// TIA Portal V17 export
// export: Created 2025-03-07T09:17:03.08606Z, ExportSetting WithDefaults, DisplayName Totally Integrated Automation Portal, DisplayVersion V17 Update 8, DisplayName TIA Portal Openness, DisplayVersion V17 Update 8, DisplayName TIA Portal Version Control Interface, DisplayVersion V17, DisplayName SINAMICS Startdrive Advanced, DisplayVersion V17 SP2, DisplayName SINAMICS Startdrive G110M, G120, G120C, G120D, G120P, G115D, DisplayVersion V17 SP2, DisplayName SINAMICS Startdrive G130, G150, S120, S150, SINAMICS MV, S210, DisplayVersion V17 SP2, DisplayName STEP 7 Professional, DisplayVersion V17 Update 8, DisplayName SINUMERIK ONE STEP 7 Toolbox, DisplayVersion V17 Update 12, DisplayName SINUMERIK 840D sl STEP 7 Toolbox, DisplayVersion V17 Update 12, DisplayName STEP 7 Safety, DisplayVersion V17 Update 6, DisplayName WinCC Advanced, DisplayVersion V17 Update 8
FUNCTION "FC7451_QUALITY_ON_DEMAND_CLADDING" : Void   // FC7451, LAD
{ S7_Optimized_Access := 'FALSE' }
AUTHOR : ETXETAR
NAME : GM-QC
VERSION : 1.0
// stored: AutoNumber false, IsIECCheckEnabled false, SetENOAutomatically false, UDAEnableTagReadback false
   VAR CONSTANT
      FC_NUMBER : DInt := 7451;
   END_VAR
   VAR_TEMP   // added for the SCL form of the ladder/FBD networks
      _w1 : Bool;
      _w2 : Bool;
   END_VAR
BEGIN

REGION Network 1: //////////_UNIT_01_//////////
END_REGION

REGION Network 2: FIXTURE 1 PART A DEMAND SET
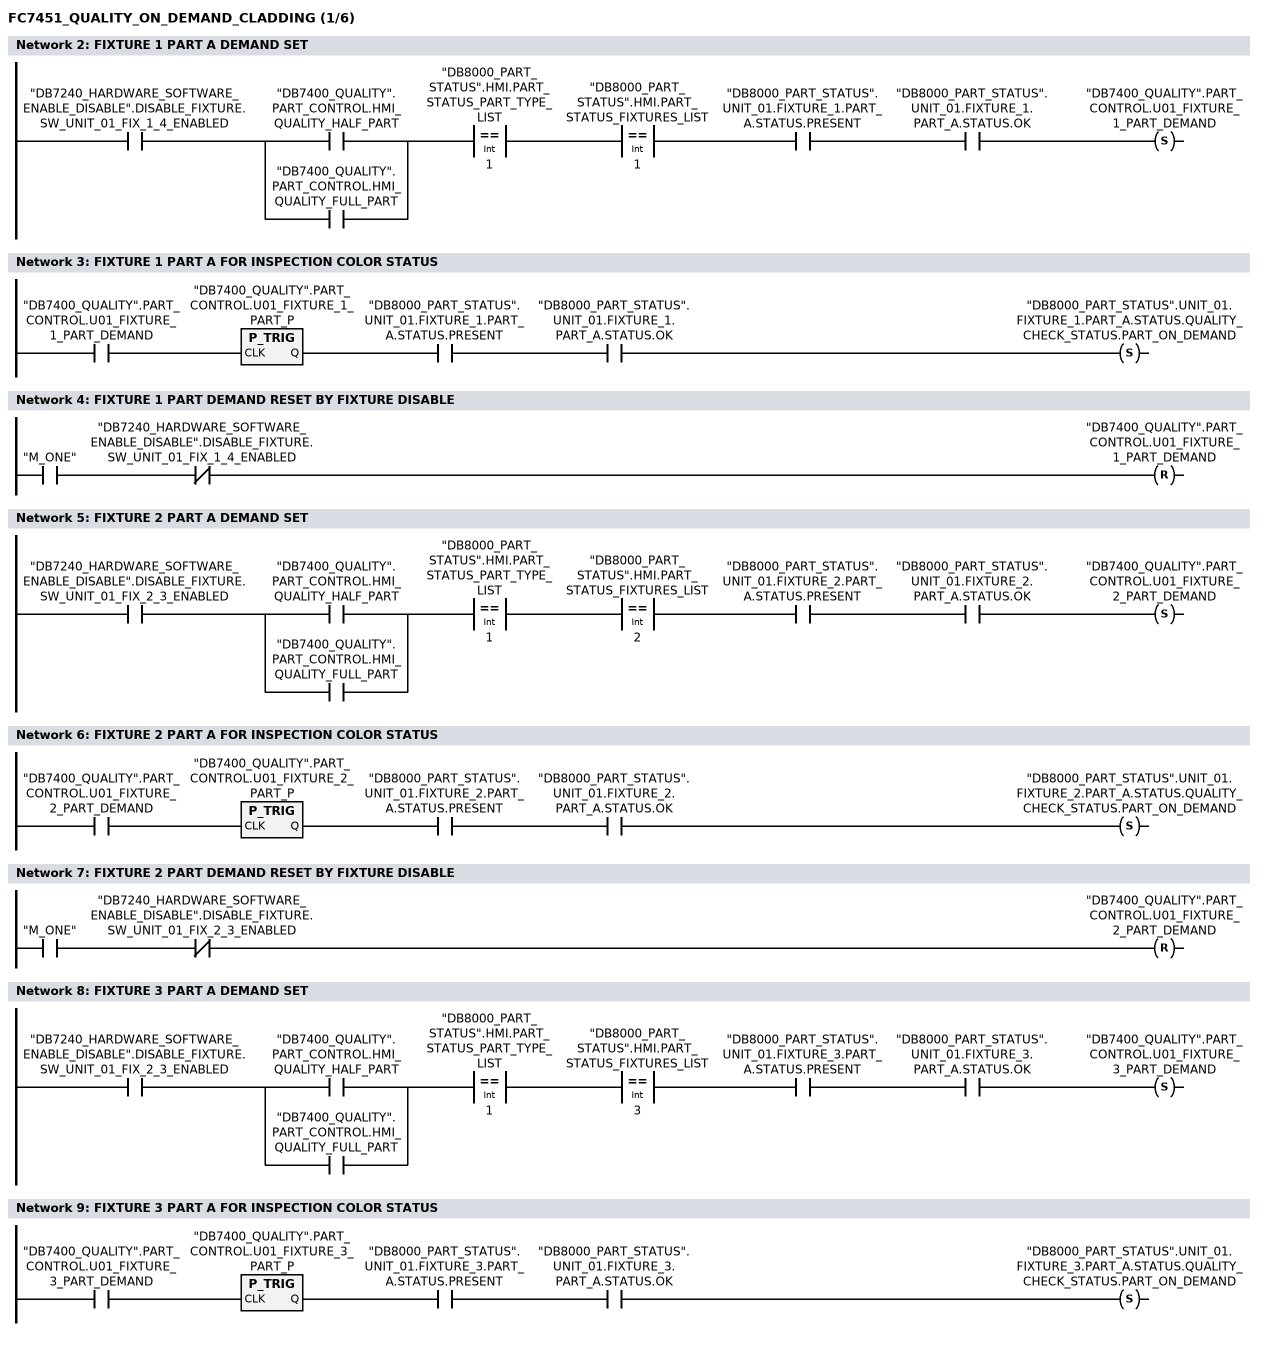
   RUNG wire#powerrail
      Contact( "DB7240_HARDWARE_SOFTWARE_ENABLE_DISABLE".DISABLE_FIXTURE.SW_UNIT_01_FIX_1_4_ENABLED )
      wire#w1
      Contact( "DB7400_QUALITY".PART_CONTROL.HMI_QUALITY_HALF_PART )
      wire#w2
      { S7_Templates := "SrcType := Int" } EQ_Contact(in1 := "DB8000_PART_STATUS".HMI.PART_STATUS_PART_TYPE_LIST, in2 := 1)
      { S7_Templates := "SrcType := Int" } EQ_Contact(in1 := "DB8000_PART_STATUS".HMI.PART_STATUS_FIXTURES_LIST, in2 := 1)
      Contact( "DB8000_PART_STATUS".UNIT_01.FIXTURE_1.PART_A.STATUS.PRESENT )
      Contact( "DB8000_PART_STATUS".UNIT_01.FIXTURE_1.PART_A.STATUS.OK )
      S_Coil( "DB7400_QUALITY".PART_CONTROL.U01_FIXTURE_1_PART_DEMAND )
   END_RUNG
   RUNG wire#w1
      Contact( "DB7400_QUALITY".PART_CONTROL.HMI_QUALITY_FULL_PART )
   END_RUNG wire#w2
   // the same network as SCL:
   IF "DB7240_HARDWARE_SOFTWARE_ENABLE_DISABLE".DISABLE_FIXTURE.SW_UNIT_01_FIX_1_4_ENABLED AND ("DB7400_QUALITY".PART_CONTROL.HMI_QUALITY_HALF_PART OR "DB7400_QUALITY".PART_CONTROL.HMI_QUALITY_FULL_PART) AND ("DB8000_PART_STATUS".HMI.PART_STATUS_PART_TYPE_LIST = 1) AND ("DB8000_PART_STATUS".HMI.PART_STATUS_FIXTURES_LIST = 1) AND "DB8000_PART_STATUS".UNIT_01.FIXTURE_1.PART_A.STATUS.PRESENT AND "DB8000_PART_STATUS".UNIT_01.FIXTURE_1.PART_A.STATUS.OK THEN
       "DB7400_QUALITY".PART_CONTROL.U01_FIXTURE_1_PART_DEMAND := TRUE;
   END_IF;
END_REGION

REGION Network 3: FIXTURE 1 PART A FOR INSPECTION COLOR STATUS
   RUNG wire#powerrail
      Contact( "DB7400_QUALITY".PART_CONTROL.U01_FIXTURE_1_PART_DEMAND )
      P_Trig( "DB7400_QUALITY".PART_CONTROL.U01_FIXTURE_1_PART_P )
      Contact( "DB8000_PART_STATUS".UNIT_01.FIXTURE_1.PART_A.STATUS.PRESENT )
      Contact( "DB8000_PART_STATUS".UNIT_01.FIXTURE_1.PART_A.STATUS.OK )
      S_Coil( "DB8000_PART_STATUS".UNIT_01.FIXTURE_1.PART_A.STATUS.QUALITY_CHECK_STATUS.PART_ON_DEMAND )
   END_RUNG
   // the same network as SCL:
   #_w1 := "DB7400_QUALITY".PART_CONTROL.U01_FIXTURE_1_PART_DEMAND AND NOT "DB7400_QUALITY".PART_CONTROL.U01_FIXTURE_1_PART_P;   // rising edge
   "DB7400_QUALITY".PART_CONTROL.U01_FIXTURE_1_PART_P := "DB7400_QUALITY".PART_CONTROL.U01_FIXTURE_1_PART_DEMAND;
   IF #_w1 AND "DB8000_PART_STATUS".UNIT_01.FIXTURE_1.PART_A.STATUS.PRESENT AND "DB8000_PART_STATUS".UNIT_01.FIXTURE_1.PART_A.STATUS.OK THEN
       "DB8000_PART_STATUS".UNIT_01.FIXTURE_1.PART_A.STATUS.QUALITY_CHECK_STATUS.PART_ON_DEMAND := TRUE;
   END_IF;
END_REGION

REGION Network 4: FIXTURE 1 PART DEMAND RESET BY FIXTURE DISABLE
   RUNG wire#powerrail
      Contact( "M_ONE" )
      I_Contact( "DB7240_HARDWARE_SOFTWARE_ENABLE_DISABLE".DISABLE_FIXTURE.SW_UNIT_01_FIX_1_4_ENABLED )
      R_Coil( "DB7400_QUALITY".PART_CONTROL.U01_FIXTURE_1_PART_DEMAND )
   END_RUNG
   // the same network as SCL:
   IF "M_ONE" AND NOT "DB7240_HARDWARE_SOFTWARE_ENABLE_DISABLE".DISABLE_FIXTURE.SW_UNIT_01_FIX_1_4_ENABLED THEN
       "DB7400_QUALITY".PART_CONTROL.U01_FIXTURE_1_PART_DEMAND := FALSE;
   END_IF;
END_REGION

REGION Network 5: FIXTURE 2 PART A DEMAND SET
   RUNG wire#powerrail
      Contact( "DB7240_HARDWARE_SOFTWARE_ENABLE_DISABLE".DISABLE_FIXTURE.SW_UNIT_01_FIX_2_3_ENABLED )
      wire#w1
      Contact( "DB7400_QUALITY".PART_CONTROL.HMI_QUALITY_HALF_PART )
      wire#w2
      { S7_Templates := "SrcType := Int" } EQ_Contact(in1 := "DB8000_PART_STATUS".HMI.PART_STATUS_PART_TYPE_LIST, in2 := 1)
      { S7_Templates := "SrcType := Int" } EQ_Contact(in1 := "DB8000_PART_STATUS".HMI.PART_STATUS_FIXTURES_LIST, in2 := 2)
      Contact( "DB8000_PART_STATUS".UNIT_01.FIXTURE_2.PART_A.STATUS.PRESENT )
      Contact( "DB8000_PART_STATUS".UNIT_01.FIXTURE_2.PART_A.STATUS.OK )
      S_Coil( "DB7400_QUALITY".PART_CONTROL.U01_FIXTURE_2_PART_DEMAND )
   END_RUNG
   RUNG wire#w1
      Contact( "DB7400_QUALITY".PART_CONTROL.HMI_QUALITY_FULL_PART )
   END_RUNG wire#w2
   // the same network as SCL:
   IF "DB7240_HARDWARE_SOFTWARE_ENABLE_DISABLE".DISABLE_FIXTURE.SW_UNIT_01_FIX_2_3_ENABLED AND ("DB7400_QUALITY".PART_CONTROL.HMI_QUALITY_HALF_PART OR "DB7400_QUALITY".PART_CONTROL.HMI_QUALITY_FULL_PART) AND ("DB8000_PART_STATUS".HMI.PART_STATUS_PART_TYPE_LIST = 1) AND ("DB8000_PART_STATUS".HMI.PART_STATUS_FIXTURES_LIST = 2) AND "DB8000_PART_STATUS".UNIT_01.FIXTURE_2.PART_A.STATUS.PRESENT AND "DB8000_PART_STATUS".UNIT_01.FIXTURE_2.PART_A.STATUS.OK THEN
       "DB7400_QUALITY".PART_CONTROL.U01_FIXTURE_2_PART_DEMAND := TRUE;
   END_IF;
END_REGION

REGION Network 6: FIXTURE 2 PART A FOR INSPECTION COLOR STATUS
   RUNG wire#powerrail
      Contact( "DB7400_QUALITY".PART_CONTROL.U01_FIXTURE_2_PART_DEMAND )
      P_Trig( "DB7400_QUALITY".PART_CONTROL.U01_FIXTURE_2_PART_P )
      Contact( "DB8000_PART_STATUS".UNIT_01.FIXTURE_2.PART_A.STATUS.PRESENT )
      Contact( "DB8000_PART_STATUS".UNIT_01.FIXTURE_2.PART_A.STATUS.OK )
      S_Coil( "DB8000_PART_STATUS".UNIT_01.FIXTURE_2.PART_A.STATUS.QUALITY_CHECK_STATUS.PART_ON_DEMAND )
   END_RUNG
   // the same network as SCL:
   #_w1 := "DB7400_QUALITY".PART_CONTROL.U01_FIXTURE_2_PART_DEMAND AND NOT "DB7400_QUALITY".PART_CONTROL.U01_FIXTURE_2_PART_P;   // rising edge
   "DB7400_QUALITY".PART_CONTROL.U01_FIXTURE_2_PART_P := "DB7400_QUALITY".PART_CONTROL.U01_FIXTURE_2_PART_DEMAND;
   IF #_w1 AND "DB8000_PART_STATUS".UNIT_01.FIXTURE_2.PART_A.STATUS.PRESENT AND "DB8000_PART_STATUS".UNIT_01.FIXTURE_2.PART_A.STATUS.OK THEN
       "DB8000_PART_STATUS".UNIT_01.FIXTURE_2.PART_A.STATUS.QUALITY_CHECK_STATUS.PART_ON_DEMAND := TRUE;
   END_IF;
END_REGION

REGION Network 7: FIXTURE 2 PART DEMAND RESET BY FIXTURE DISABLE
   RUNG wire#powerrail
      Contact( "M_ONE" )
      I_Contact( "DB7240_HARDWARE_SOFTWARE_ENABLE_DISABLE".DISABLE_FIXTURE.SW_UNIT_01_FIX_2_3_ENABLED )
      R_Coil( "DB7400_QUALITY".PART_CONTROL.U01_FIXTURE_2_PART_DEMAND )
   END_RUNG
   // the same network as SCL:
   IF "M_ONE" AND NOT "DB7240_HARDWARE_SOFTWARE_ENABLE_DISABLE".DISABLE_FIXTURE.SW_UNIT_01_FIX_2_3_ENABLED THEN
       "DB7400_QUALITY".PART_CONTROL.U01_FIXTURE_2_PART_DEMAND := FALSE;
   END_IF;
END_REGION

REGION Network 8: FIXTURE 3 PART A DEMAND SET
   RUNG wire#powerrail
      Contact( "DB7240_HARDWARE_SOFTWARE_ENABLE_DISABLE".DISABLE_FIXTURE.SW_UNIT_01_FIX_2_3_ENABLED )
      wire#w1
      Contact( "DB7400_QUALITY".PART_CONTROL.HMI_QUALITY_HALF_PART )
      wire#w2
      { S7_Templates := "SrcType := Int" } EQ_Contact(in1 := "DB8000_PART_STATUS".HMI.PART_STATUS_PART_TYPE_LIST, in2 := 1)
      { S7_Templates := "SrcType := Int" } EQ_Contact(in1 := "DB8000_PART_STATUS".HMI.PART_STATUS_FIXTURES_LIST, in2 := 3)
      Contact( "DB8000_PART_STATUS".UNIT_01.FIXTURE_3.PART_A.STATUS.PRESENT )
      Contact( "DB8000_PART_STATUS".UNIT_01.FIXTURE_3.PART_A.STATUS.OK )
      S_Coil( "DB7400_QUALITY".PART_CONTROL.U01_FIXTURE_3_PART_DEMAND )
   END_RUNG
   RUNG wire#w1
      Contact( "DB7400_QUALITY".PART_CONTROL.HMI_QUALITY_FULL_PART )
   END_RUNG wire#w2
   // the same network as SCL:
   IF "DB7240_HARDWARE_SOFTWARE_ENABLE_DISABLE".DISABLE_FIXTURE.SW_UNIT_01_FIX_2_3_ENABLED AND ("DB7400_QUALITY".PART_CONTROL.HMI_QUALITY_HALF_PART OR "DB7400_QUALITY".PART_CONTROL.HMI_QUALITY_FULL_PART) AND ("DB8000_PART_STATUS".HMI.PART_STATUS_PART_TYPE_LIST = 1) AND ("DB8000_PART_STATUS".HMI.PART_STATUS_FIXTURES_LIST = 3) AND "DB8000_PART_STATUS".UNIT_01.FIXTURE_3.PART_A.STATUS.PRESENT AND "DB8000_PART_STATUS".UNIT_01.FIXTURE_3.PART_A.STATUS.OK THEN
       "DB7400_QUALITY".PART_CONTROL.U01_FIXTURE_3_PART_DEMAND := TRUE;
   END_IF;
END_REGION

REGION Network 9: FIXTURE 3 PART A FOR INSPECTION COLOR STATUS
   RUNG wire#powerrail
      Contact( "DB7400_QUALITY".PART_CONTROL.U01_FIXTURE_3_PART_DEMAND )
      P_Trig( "DB7400_QUALITY".PART_CONTROL.U01_FIXTURE_3_PART_P )
      Contact( "DB8000_PART_STATUS".UNIT_01.FIXTURE_3.PART_A.STATUS.PRESENT )
      Contact( "DB8000_PART_STATUS".UNIT_01.FIXTURE_3.PART_A.STATUS.OK )
      S_Coil( "DB8000_PART_STATUS".UNIT_01.FIXTURE_3.PART_A.STATUS.QUALITY_CHECK_STATUS.PART_ON_DEMAND )
   END_RUNG
   // the same network as SCL:
   #_w1 := "DB7400_QUALITY".PART_CONTROL.U01_FIXTURE_3_PART_DEMAND AND NOT "DB7400_QUALITY".PART_CONTROL.U01_FIXTURE_3_PART_P;   // rising edge
   "DB7400_QUALITY".PART_CONTROL.U01_FIXTURE_3_PART_P := "DB7400_QUALITY".PART_CONTROL.U01_FIXTURE_3_PART_DEMAND;
   IF #_w1 AND "DB8000_PART_STATUS".UNIT_01.FIXTURE_3.PART_A.STATUS.PRESENT AND "DB8000_PART_STATUS".UNIT_01.FIXTURE_3.PART_A.STATUS.OK THEN
       "DB8000_PART_STATUS".UNIT_01.FIXTURE_3.PART_A.STATUS.QUALITY_CHECK_STATUS.PART_ON_DEMAND := TRUE;
   END_IF;
END_REGION

REGION Network 10: FIXTURE 3 PART DEMAND RESET BY FIXTURE DISABLE
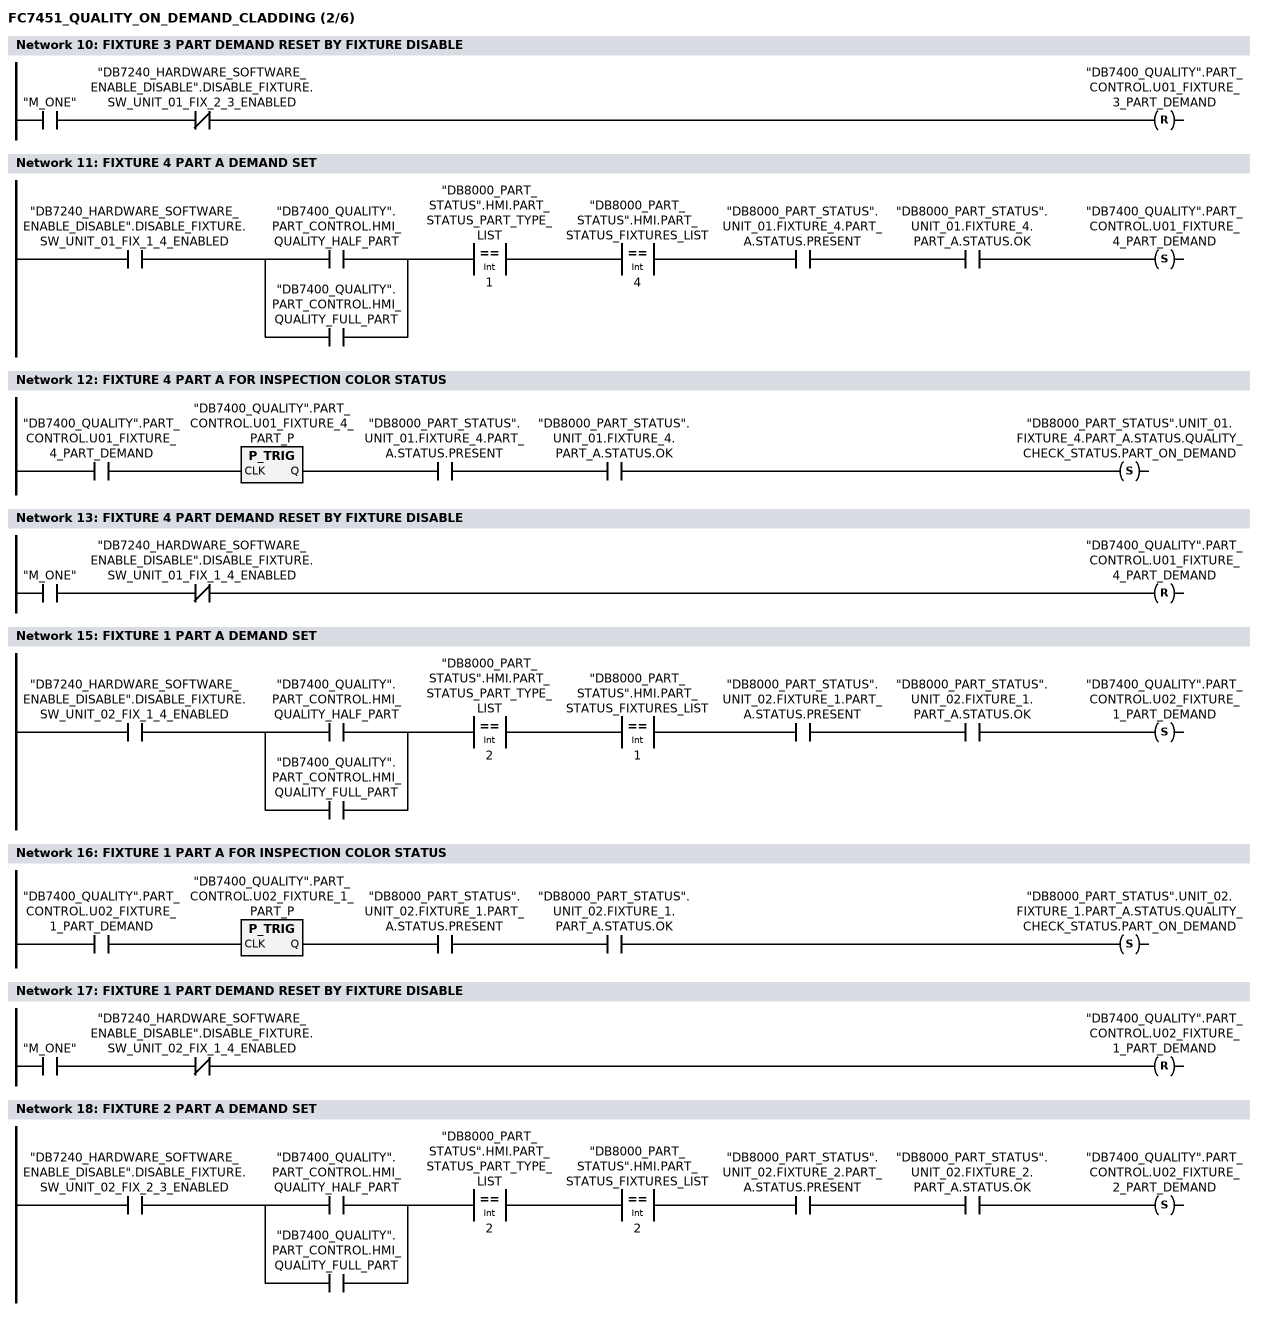
   RUNG wire#powerrail
      Contact( "M_ONE" )
      I_Contact( "DB7240_HARDWARE_SOFTWARE_ENABLE_DISABLE".DISABLE_FIXTURE.SW_UNIT_01_FIX_2_3_ENABLED )
      R_Coil( "DB7400_QUALITY".PART_CONTROL.U01_FIXTURE_3_PART_DEMAND )
   END_RUNG
   // the same network as SCL:
   IF "M_ONE" AND NOT "DB7240_HARDWARE_SOFTWARE_ENABLE_DISABLE".DISABLE_FIXTURE.SW_UNIT_01_FIX_2_3_ENABLED THEN
       "DB7400_QUALITY".PART_CONTROL.U01_FIXTURE_3_PART_DEMAND := FALSE;
   END_IF;
END_REGION

REGION Network 11: FIXTURE 4 PART A DEMAND SET
   RUNG wire#powerrail
      Contact( "DB7240_HARDWARE_SOFTWARE_ENABLE_DISABLE".DISABLE_FIXTURE.SW_UNIT_01_FIX_1_4_ENABLED )
      wire#w1
      Contact( "DB7400_QUALITY".PART_CONTROL.HMI_QUALITY_HALF_PART )
      wire#w2
      { S7_Templates := "SrcType := Int" } EQ_Contact(in1 := "DB8000_PART_STATUS".HMI.PART_STATUS_PART_TYPE_LIST, in2 := 1)
      { S7_Templates := "SrcType := Int" } EQ_Contact(in1 := "DB8000_PART_STATUS".HMI.PART_STATUS_FIXTURES_LIST, in2 := 4)
      Contact( "DB8000_PART_STATUS".UNIT_01.FIXTURE_4.PART_A.STATUS.PRESENT )
      Contact( "DB8000_PART_STATUS".UNIT_01.FIXTURE_4.PART_A.STATUS.OK )
      S_Coil( "DB7400_QUALITY".PART_CONTROL.U01_FIXTURE_4_PART_DEMAND )
   END_RUNG
   RUNG wire#w1
      Contact( "DB7400_QUALITY".PART_CONTROL.HMI_QUALITY_FULL_PART )
   END_RUNG wire#w2
   // the same network as SCL:
   IF "DB7240_HARDWARE_SOFTWARE_ENABLE_DISABLE".DISABLE_FIXTURE.SW_UNIT_01_FIX_1_4_ENABLED AND ("DB7400_QUALITY".PART_CONTROL.HMI_QUALITY_HALF_PART OR "DB7400_QUALITY".PART_CONTROL.HMI_QUALITY_FULL_PART) AND ("DB8000_PART_STATUS".HMI.PART_STATUS_PART_TYPE_LIST = 1) AND ("DB8000_PART_STATUS".HMI.PART_STATUS_FIXTURES_LIST = 4) AND "DB8000_PART_STATUS".UNIT_01.FIXTURE_4.PART_A.STATUS.PRESENT AND "DB8000_PART_STATUS".UNIT_01.FIXTURE_4.PART_A.STATUS.OK THEN
       "DB7400_QUALITY".PART_CONTROL.U01_FIXTURE_4_PART_DEMAND := TRUE;
   END_IF;
END_REGION

REGION Network 12: FIXTURE 4 PART A FOR INSPECTION COLOR STATUS
   RUNG wire#powerrail
      Contact( "DB7400_QUALITY".PART_CONTROL.U01_FIXTURE_4_PART_DEMAND )
      P_Trig( "DB7400_QUALITY".PART_CONTROL.U01_FIXTURE_4_PART_P )
      Contact( "DB8000_PART_STATUS".UNIT_01.FIXTURE_4.PART_A.STATUS.PRESENT )
      Contact( "DB8000_PART_STATUS".UNIT_01.FIXTURE_4.PART_A.STATUS.OK )
      S_Coil( "DB8000_PART_STATUS".UNIT_01.FIXTURE_4.PART_A.STATUS.QUALITY_CHECK_STATUS.PART_ON_DEMAND )
   END_RUNG
   // the same network as SCL:
   #_w1 := "DB7400_QUALITY".PART_CONTROL.U01_FIXTURE_4_PART_DEMAND AND NOT "DB7400_QUALITY".PART_CONTROL.U01_FIXTURE_4_PART_P;   // rising edge
   "DB7400_QUALITY".PART_CONTROL.U01_FIXTURE_4_PART_P := "DB7400_QUALITY".PART_CONTROL.U01_FIXTURE_4_PART_DEMAND;
   IF #_w1 AND "DB8000_PART_STATUS".UNIT_01.FIXTURE_4.PART_A.STATUS.PRESENT AND "DB8000_PART_STATUS".UNIT_01.FIXTURE_4.PART_A.STATUS.OK THEN
       "DB8000_PART_STATUS".UNIT_01.FIXTURE_4.PART_A.STATUS.QUALITY_CHECK_STATUS.PART_ON_DEMAND := TRUE;
   END_IF;
END_REGION

REGION Network 13: FIXTURE 4 PART DEMAND RESET BY FIXTURE DISABLE
   RUNG wire#powerrail
      Contact( "M_ONE" )
      I_Contact( "DB7240_HARDWARE_SOFTWARE_ENABLE_DISABLE".DISABLE_FIXTURE.SW_UNIT_01_FIX_1_4_ENABLED )
      R_Coil( "DB7400_QUALITY".PART_CONTROL.U01_FIXTURE_4_PART_DEMAND )
   END_RUNG
   // the same network as SCL:
   IF "M_ONE" AND NOT "DB7240_HARDWARE_SOFTWARE_ENABLE_DISABLE".DISABLE_FIXTURE.SW_UNIT_01_FIX_1_4_ENABLED THEN
       "DB7400_QUALITY".PART_CONTROL.U01_FIXTURE_4_PART_DEMAND := FALSE;
   END_IF;
END_REGION

REGION Network 14: //////////_UNIT_02_//////////
END_REGION

REGION Network 15: FIXTURE 1 PART A DEMAND SET
   RUNG wire#powerrail
      Contact( "DB7240_HARDWARE_SOFTWARE_ENABLE_DISABLE".DISABLE_FIXTURE.SW_UNIT_02_FIX_1_4_ENABLED )
      wire#w1
      Contact( "DB7400_QUALITY".PART_CONTROL.HMI_QUALITY_HALF_PART )
      wire#w2
      { S7_Templates := "SrcType := Int" } EQ_Contact(in1 := "DB8000_PART_STATUS".HMI.PART_STATUS_PART_TYPE_LIST, in2 := 2)
      { S7_Templates := "SrcType := Int" } EQ_Contact(in1 := "DB8000_PART_STATUS".HMI.PART_STATUS_FIXTURES_LIST, in2 := 1)
      Contact( "DB8000_PART_STATUS".UNIT_02.FIXTURE_1.PART_A.STATUS.PRESENT )
      Contact( "DB8000_PART_STATUS".UNIT_02.FIXTURE_1.PART_A.STATUS.OK )
      S_Coil( "DB7400_QUALITY".PART_CONTROL.U02_FIXTURE_1_PART_DEMAND )
   END_RUNG
   RUNG wire#w1
      Contact( "DB7400_QUALITY".PART_CONTROL.HMI_QUALITY_FULL_PART )
   END_RUNG wire#w2
   // the same network as SCL:
   IF "DB7240_HARDWARE_SOFTWARE_ENABLE_DISABLE".DISABLE_FIXTURE.SW_UNIT_02_FIX_1_4_ENABLED AND ("DB7400_QUALITY".PART_CONTROL.HMI_QUALITY_HALF_PART OR "DB7400_QUALITY".PART_CONTROL.HMI_QUALITY_FULL_PART) AND ("DB8000_PART_STATUS".HMI.PART_STATUS_PART_TYPE_LIST = 2) AND ("DB8000_PART_STATUS".HMI.PART_STATUS_FIXTURES_LIST = 1) AND "DB8000_PART_STATUS".UNIT_02.FIXTURE_1.PART_A.STATUS.PRESENT AND "DB8000_PART_STATUS".UNIT_02.FIXTURE_1.PART_A.STATUS.OK THEN
       "DB7400_QUALITY".PART_CONTROL.U02_FIXTURE_1_PART_DEMAND := TRUE;
   END_IF;
END_REGION

REGION Network 16: FIXTURE 1 PART A FOR INSPECTION COLOR STATUS
   RUNG wire#powerrail
      Contact( "DB7400_QUALITY".PART_CONTROL.U02_FIXTURE_1_PART_DEMAND )
      P_Trig( "DB7400_QUALITY".PART_CONTROL.U02_FIXTURE_1_PART_P )
      Contact( "DB8000_PART_STATUS".UNIT_02.FIXTURE_1.PART_A.STATUS.PRESENT )
      Contact( "DB8000_PART_STATUS".UNIT_02.FIXTURE_1.PART_A.STATUS.OK )
      S_Coil( "DB8000_PART_STATUS".UNIT_02.FIXTURE_1.PART_A.STATUS.QUALITY_CHECK_STATUS.PART_ON_DEMAND )
   END_RUNG
   // the same network as SCL:
   #_w1 := "DB7400_QUALITY".PART_CONTROL.U02_FIXTURE_1_PART_DEMAND AND NOT "DB7400_QUALITY".PART_CONTROL.U02_FIXTURE_1_PART_P;   // rising edge
   "DB7400_QUALITY".PART_CONTROL.U02_FIXTURE_1_PART_P := "DB7400_QUALITY".PART_CONTROL.U02_FIXTURE_1_PART_DEMAND;
   IF #_w1 AND "DB8000_PART_STATUS".UNIT_02.FIXTURE_1.PART_A.STATUS.PRESENT AND "DB8000_PART_STATUS".UNIT_02.FIXTURE_1.PART_A.STATUS.OK THEN
       "DB8000_PART_STATUS".UNIT_02.FIXTURE_1.PART_A.STATUS.QUALITY_CHECK_STATUS.PART_ON_DEMAND := TRUE;
   END_IF;
END_REGION

REGION Network 17: FIXTURE 1 PART DEMAND RESET BY FIXTURE DISABLE
   RUNG wire#powerrail
      Contact( "M_ONE" )
      I_Contact( "DB7240_HARDWARE_SOFTWARE_ENABLE_DISABLE".DISABLE_FIXTURE.SW_UNIT_02_FIX_1_4_ENABLED )
      R_Coil( "DB7400_QUALITY".PART_CONTROL.U02_FIXTURE_1_PART_DEMAND )
   END_RUNG
   // the same network as SCL:
   IF "M_ONE" AND NOT "DB7240_HARDWARE_SOFTWARE_ENABLE_DISABLE".DISABLE_FIXTURE.SW_UNIT_02_FIX_1_4_ENABLED THEN
       "DB7400_QUALITY".PART_CONTROL.U02_FIXTURE_1_PART_DEMAND := FALSE;
   END_IF;
END_REGION

REGION Network 18: FIXTURE 2 PART A DEMAND SET
   RUNG wire#powerrail
      Contact( "DB7240_HARDWARE_SOFTWARE_ENABLE_DISABLE".DISABLE_FIXTURE.SW_UNIT_02_FIX_2_3_ENABLED )
      wire#w1
      Contact( "DB7400_QUALITY".PART_CONTROL.HMI_QUALITY_HALF_PART )
      wire#w2
      { S7_Templates := "SrcType := Int" } EQ_Contact(in1 := "DB8000_PART_STATUS".HMI.PART_STATUS_PART_TYPE_LIST, in2 := 2)
      { S7_Templates := "SrcType := Int" } EQ_Contact(in1 := "DB8000_PART_STATUS".HMI.PART_STATUS_FIXTURES_LIST, in2 := 2)
      Contact( "DB8000_PART_STATUS".UNIT_02.FIXTURE_2.PART_A.STATUS.PRESENT )
      Contact( "DB8000_PART_STATUS".UNIT_02.FIXTURE_2.PART_A.STATUS.OK )
      S_Coil( "DB7400_QUALITY".PART_CONTROL.U02_FIXTURE_2_PART_DEMAND )
   END_RUNG
   RUNG wire#w1
      Contact( "DB7400_QUALITY".PART_CONTROL.HMI_QUALITY_FULL_PART )
   END_RUNG wire#w2
   // the same network as SCL:
   IF "DB7240_HARDWARE_SOFTWARE_ENABLE_DISABLE".DISABLE_FIXTURE.SW_UNIT_02_FIX_2_3_ENABLED AND ("DB7400_QUALITY".PART_CONTROL.HMI_QUALITY_HALF_PART OR "DB7400_QUALITY".PART_CONTROL.HMI_QUALITY_FULL_PART) AND ("DB8000_PART_STATUS".HMI.PART_STATUS_PART_TYPE_LIST = 2) AND ("DB8000_PART_STATUS".HMI.PART_STATUS_FIXTURES_LIST = 2) AND "DB8000_PART_STATUS".UNIT_02.FIXTURE_2.PART_A.STATUS.PRESENT AND "DB8000_PART_STATUS".UNIT_02.FIXTURE_2.PART_A.STATUS.OK THEN
       "DB7400_QUALITY".PART_CONTROL.U02_FIXTURE_2_PART_DEMAND := TRUE;
   END_IF;
END_REGION

REGION Network 19: FIXTURE 2 PART A FOR INSPECTION COLOR STATUS
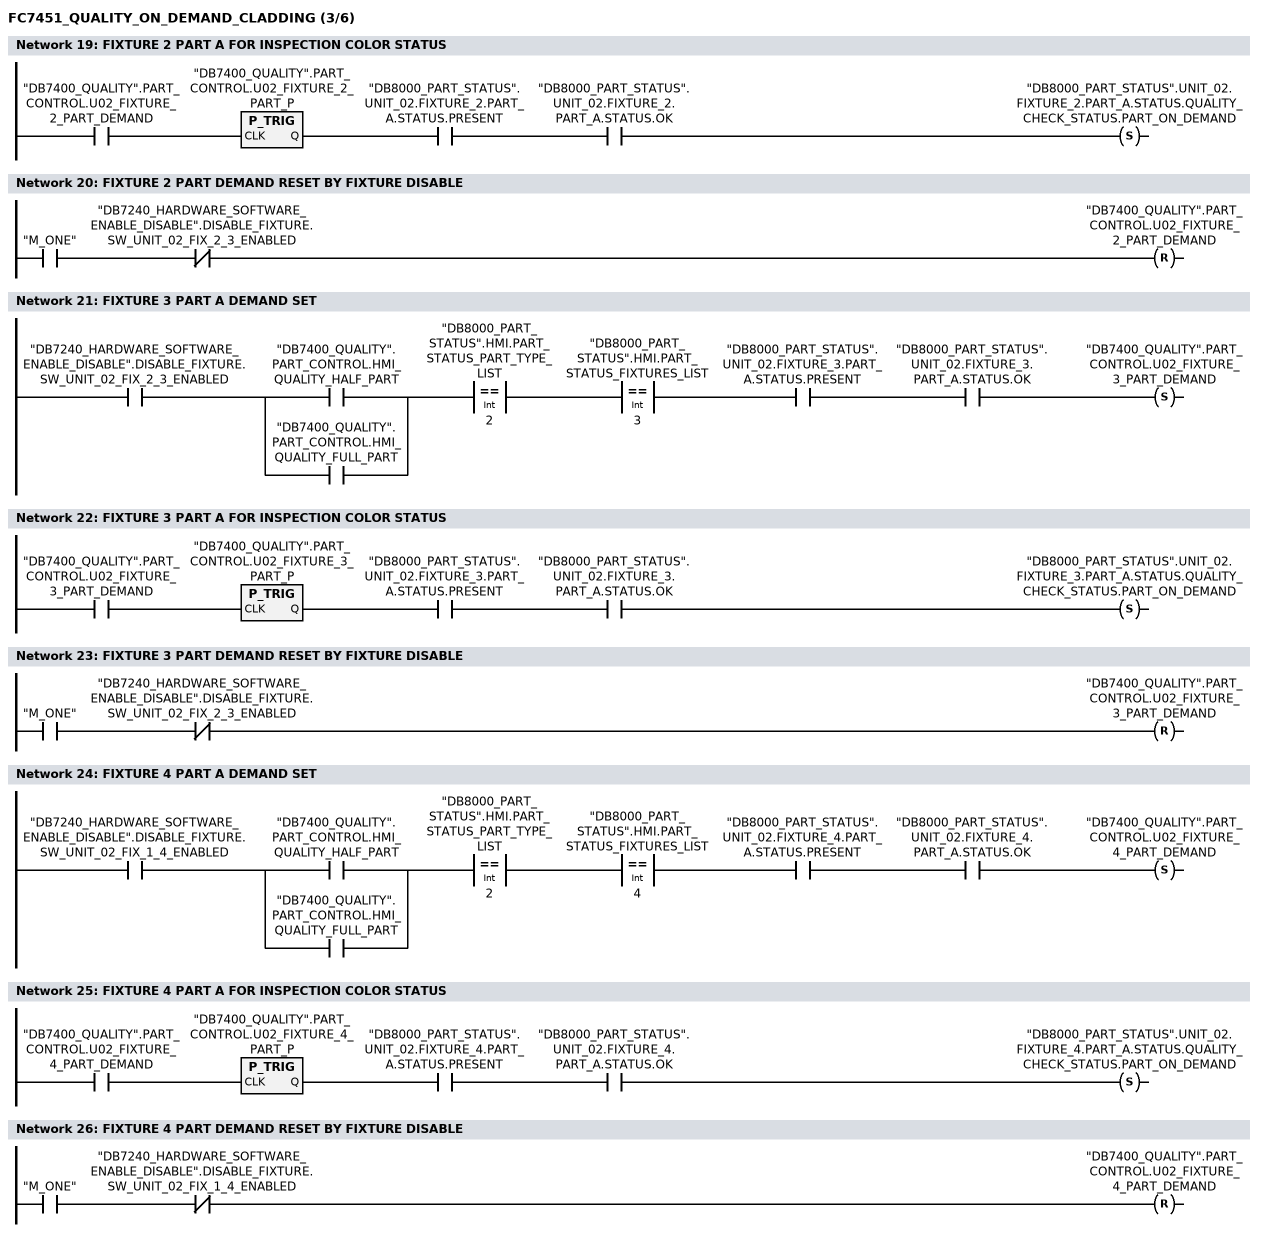
   RUNG wire#powerrail
      Contact( "DB7400_QUALITY".PART_CONTROL.U02_FIXTURE_2_PART_DEMAND )
      P_Trig( "DB7400_QUALITY".PART_CONTROL.U02_FIXTURE_2_PART_P )
      Contact( "DB8000_PART_STATUS".UNIT_02.FIXTURE_2.PART_A.STATUS.PRESENT )
      Contact( "DB8000_PART_STATUS".UNIT_02.FIXTURE_2.PART_A.STATUS.OK )
      S_Coil( "DB8000_PART_STATUS".UNIT_02.FIXTURE_2.PART_A.STATUS.QUALITY_CHECK_STATUS.PART_ON_DEMAND )
   END_RUNG
   // the same network as SCL:
   #_w1 := "DB7400_QUALITY".PART_CONTROL.U02_FIXTURE_2_PART_DEMAND AND NOT "DB7400_QUALITY".PART_CONTROL.U02_FIXTURE_2_PART_P;   // rising edge
   "DB7400_QUALITY".PART_CONTROL.U02_FIXTURE_2_PART_P := "DB7400_QUALITY".PART_CONTROL.U02_FIXTURE_2_PART_DEMAND;
   IF #_w1 AND "DB8000_PART_STATUS".UNIT_02.FIXTURE_2.PART_A.STATUS.PRESENT AND "DB8000_PART_STATUS".UNIT_02.FIXTURE_2.PART_A.STATUS.OK THEN
       "DB8000_PART_STATUS".UNIT_02.FIXTURE_2.PART_A.STATUS.QUALITY_CHECK_STATUS.PART_ON_DEMAND := TRUE;
   END_IF;
END_REGION

REGION Network 20: FIXTURE 2 PART DEMAND RESET BY FIXTURE DISABLE
   RUNG wire#powerrail
      Contact( "M_ONE" )
      I_Contact( "DB7240_HARDWARE_SOFTWARE_ENABLE_DISABLE".DISABLE_FIXTURE.SW_UNIT_02_FIX_2_3_ENABLED )
      R_Coil( "DB7400_QUALITY".PART_CONTROL.U02_FIXTURE_2_PART_DEMAND )
   END_RUNG
   // the same network as SCL:
   IF "M_ONE" AND NOT "DB7240_HARDWARE_SOFTWARE_ENABLE_DISABLE".DISABLE_FIXTURE.SW_UNIT_02_FIX_2_3_ENABLED THEN
       "DB7400_QUALITY".PART_CONTROL.U02_FIXTURE_2_PART_DEMAND := FALSE;
   END_IF;
END_REGION

REGION Network 21: FIXTURE 3 PART A DEMAND SET
   RUNG wire#powerrail
      Contact( "DB7240_HARDWARE_SOFTWARE_ENABLE_DISABLE".DISABLE_FIXTURE.SW_UNIT_02_FIX_2_3_ENABLED )
      wire#w1
      Contact( "DB7400_QUALITY".PART_CONTROL.HMI_QUALITY_HALF_PART )
      wire#w2
      { S7_Templates := "SrcType := Int" } EQ_Contact(in1 := "DB8000_PART_STATUS".HMI.PART_STATUS_PART_TYPE_LIST, in2 := 2)
      { S7_Templates := "SrcType := Int" } EQ_Contact(in1 := "DB8000_PART_STATUS".HMI.PART_STATUS_FIXTURES_LIST, in2 := 3)
      Contact( "DB8000_PART_STATUS".UNIT_02.FIXTURE_3.PART_A.STATUS.PRESENT )
      Contact( "DB8000_PART_STATUS".UNIT_02.FIXTURE_3.PART_A.STATUS.OK )
      S_Coil( "DB7400_QUALITY".PART_CONTROL.U02_FIXTURE_3_PART_DEMAND )
   END_RUNG
   RUNG wire#w1
      Contact( "DB7400_QUALITY".PART_CONTROL.HMI_QUALITY_FULL_PART )
   END_RUNG wire#w2
   // the same network as SCL:
   IF "DB7240_HARDWARE_SOFTWARE_ENABLE_DISABLE".DISABLE_FIXTURE.SW_UNIT_02_FIX_2_3_ENABLED AND ("DB7400_QUALITY".PART_CONTROL.HMI_QUALITY_HALF_PART OR "DB7400_QUALITY".PART_CONTROL.HMI_QUALITY_FULL_PART) AND ("DB8000_PART_STATUS".HMI.PART_STATUS_PART_TYPE_LIST = 2) AND ("DB8000_PART_STATUS".HMI.PART_STATUS_FIXTURES_LIST = 3) AND "DB8000_PART_STATUS".UNIT_02.FIXTURE_3.PART_A.STATUS.PRESENT AND "DB8000_PART_STATUS".UNIT_02.FIXTURE_3.PART_A.STATUS.OK THEN
       "DB7400_QUALITY".PART_CONTROL.U02_FIXTURE_3_PART_DEMAND := TRUE;
   END_IF;
END_REGION

REGION Network 22: FIXTURE 3 PART A FOR INSPECTION COLOR STATUS
   RUNG wire#powerrail
      Contact( "DB7400_QUALITY".PART_CONTROL.U02_FIXTURE_3_PART_DEMAND )
      P_Trig( "DB7400_QUALITY".PART_CONTROL.U02_FIXTURE_3_PART_P )
      Contact( "DB8000_PART_STATUS".UNIT_02.FIXTURE_3.PART_A.STATUS.PRESENT )
      Contact( "DB8000_PART_STATUS".UNIT_02.FIXTURE_3.PART_A.STATUS.OK )
      S_Coil( "DB8000_PART_STATUS".UNIT_02.FIXTURE_3.PART_A.STATUS.QUALITY_CHECK_STATUS.PART_ON_DEMAND )
   END_RUNG
   // the same network as SCL:
   #_w1 := "DB7400_QUALITY".PART_CONTROL.U02_FIXTURE_3_PART_DEMAND AND NOT "DB7400_QUALITY".PART_CONTROL.U02_FIXTURE_3_PART_P;   // rising edge
   "DB7400_QUALITY".PART_CONTROL.U02_FIXTURE_3_PART_P := "DB7400_QUALITY".PART_CONTROL.U02_FIXTURE_3_PART_DEMAND;
   IF #_w1 AND "DB8000_PART_STATUS".UNIT_02.FIXTURE_3.PART_A.STATUS.PRESENT AND "DB8000_PART_STATUS".UNIT_02.FIXTURE_3.PART_A.STATUS.OK THEN
       "DB8000_PART_STATUS".UNIT_02.FIXTURE_3.PART_A.STATUS.QUALITY_CHECK_STATUS.PART_ON_DEMAND := TRUE;
   END_IF;
END_REGION

REGION Network 23: FIXTURE 3 PART DEMAND RESET BY FIXTURE DISABLE
   RUNG wire#powerrail
      Contact( "M_ONE" )
      I_Contact( "DB7240_HARDWARE_SOFTWARE_ENABLE_DISABLE".DISABLE_FIXTURE.SW_UNIT_02_FIX_2_3_ENABLED )
      R_Coil( "DB7400_QUALITY".PART_CONTROL.U02_FIXTURE_3_PART_DEMAND )
   END_RUNG
   // the same network as SCL:
   IF "M_ONE" AND NOT "DB7240_HARDWARE_SOFTWARE_ENABLE_DISABLE".DISABLE_FIXTURE.SW_UNIT_02_FIX_2_3_ENABLED THEN
       "DB7400_QUALITY".PART_CONTROL.U02_FIXTURE_3_PART_DEMAND := FALSE;
   END_IF;
END_REGION

REGION Network 24: FIXTURE 4 PART A DEMAND SET
   RUNG wire#powerrail
      Contact( "DB7240_HARDWARE_SOFTWARE_ENABLE_DISABLE".DISABLE_FIXTURE.SW_UNIT_02_FIX_1_4_ENABLED )
      wire#w1
      Contact( "DB7400_QUALITY".PART_CONTROL.HMI_QUALITY_HALF_PART )
      wire#w2
      { S7_Templates := "SrcType := Int" } EQ_Contact(in1 := "DB8000_PART_STATUS".HMI.PART_STATUS_PART_TYPE_LIST, in2 := 2)
      { S7_Templates := "SrcType := Int" } EQ_Contact(in1 := "DB8000_PART_STATUS".HMI.PART_STATUS_FIXTURES_LIST, in2 := 4)
      Contact( "DB8000_PART_STATUS".UNIT_02.FIXTURE_4.PART_A.STATUS.PRESENT )
      Contact( "DB8000_PART_STATUS".UNIT_02.FIXTURE_4.PART_A.STATUS.OK )
      S_Coil( "DB7400_QUALITY".PART_CONTROL.U02_FIXTURE_4_PART_DEMAND )
   END_RUNG
   RUNG wire#w1
      Contact( "DB7400_QUALITY".PART_CONTROL.HMI_QUALITY_FULL_PART )
   END_RUNG wire#w2
   // the same network as SCL:
   IF "DB7240_HARDWARE_SOFTWARE_ENABLE_DISABLE".DISABLE_FIXTURE.SW_UNIT_02_FIX_1_4_ENABLED AND ("DB7400_QUALITY".PART_CONTROL.HMI_QUALITY_HALF_PART OR "DB7400_QUALITY".PART_CONTROL.HMI_QUALITY_FULL_PART) AND ("DB8000_PART_STATUS".HMI.PART_STATUS_PART_TYPE_LIST = 2) AND ("DB8000_PART_STATUS".HMI.PART_STATUS_FIXTURES_LIST = 4) AND "DB8000_PART_STATUS".UNIT_02.FIXTURE_4.PART_A.STATUS.PRESENT AND "DB8000_PART_STATUS".UNIT_02.FIXTURE_4.PART_A.STATUS.OK THEN
       "DB7400_QUALITY".PART_CONTROL.U02_FIXTURE_4_PART_DEMAND := TRUE;
   END_IF;
END_REGION

REGION Network 25: FIXTURE 4 PART A FOR INSPECTION COLOR STATUS
   RUNG wire#powerrail
      Contact( "DB7400_QUALITY".PART_CONTROL.U02_FIXTURE_4_PART_DEMAND )
      P_Trig( "DB7400_QUALITY".PART_CONTROL.U02_FIXTURE_4_PART_P )
      Contact( "DB8000_PART_STATUS".UNIT_02.FIXTURE_4.PART_A.STATUS.PRESENT )
      Contact( "DB8000_PART_STATUS".UNIT_02.FIXTURE_4.PART_A.STATUS.OK )
      S_Coil( "DB8000_PART_STATUS".UNIT_02.FIXTURE_4.PART_A.STATUS.QUALITY_CHECK_STATUS.PART_ON_DEMAND )
   END_RUNG
   // the same network as SCL:
   #_w1 := "DB7400_QUALITY".PART_CONTROL.U02_FIXTURE_4_PART_DEMAND AND NOT "DB7400_QUALITY".PART_CONTROL.U02_FIXTURE_4_PART_P;   // rising edge
   "DB7400_QUALITY".PART_CONTROL.U02_FIXTURE_4_PART_P := "DB7400_QUALITY".PART_CONTROL.U02_FIXTURE_4_PART_DEMAND;
   IF #_w1 AND "DB8000_PART_STATUS".UNIT_02.FIXTURE_4.PART_A.STATUS.PRESENT AND "DB8000_PART_STATUS".UNIT_02.FIXTURE_4.PART_A.STATUS.OK THEN
       "DB8000_PART_STATUS".UNIT_02.FIXTURE_4.PART_A.STATUS.QUALITY_CHECK_STATUS.PART_ON_DEMAND := TRUE;
   END_IF;
END_REGION

REGION Network 26: FIXTURE 4 PART DEMAND RESET BY FIXTURE DISABLE
   RUNG wire#powerrail
      Contact( "M_ONE" )
      I_Contact( "DB7240_HARDWARE_SOFTWARE_ENABLE_DISABLE".DISABLE_FIXTURE.SW_UNIT_02_FIX_1_4_ENABLED )
      R_Coil( "DB7400_QUALITY".PART_CONTROL.U02_FIXTURE_4_PART_DEMAND )
   END_RUNG
   // the same network as SCL:
   IF "M_ONE" AND NOT "DB7240_HARDWARE_SOFTWARE_ENABLE_DISABLE".DISABLE_FIXTURE.SW_UNIT_02_FIX_1_4_ENABLED THEN
       "DB7400_QUALITY".PART_CONTROL.U02_FIXTURE_4_PART_DEMAND := FALSE;
   END_IF;
END_REGION

REGION Network 27: PART DEMAND RESET CANCEL BUTTON
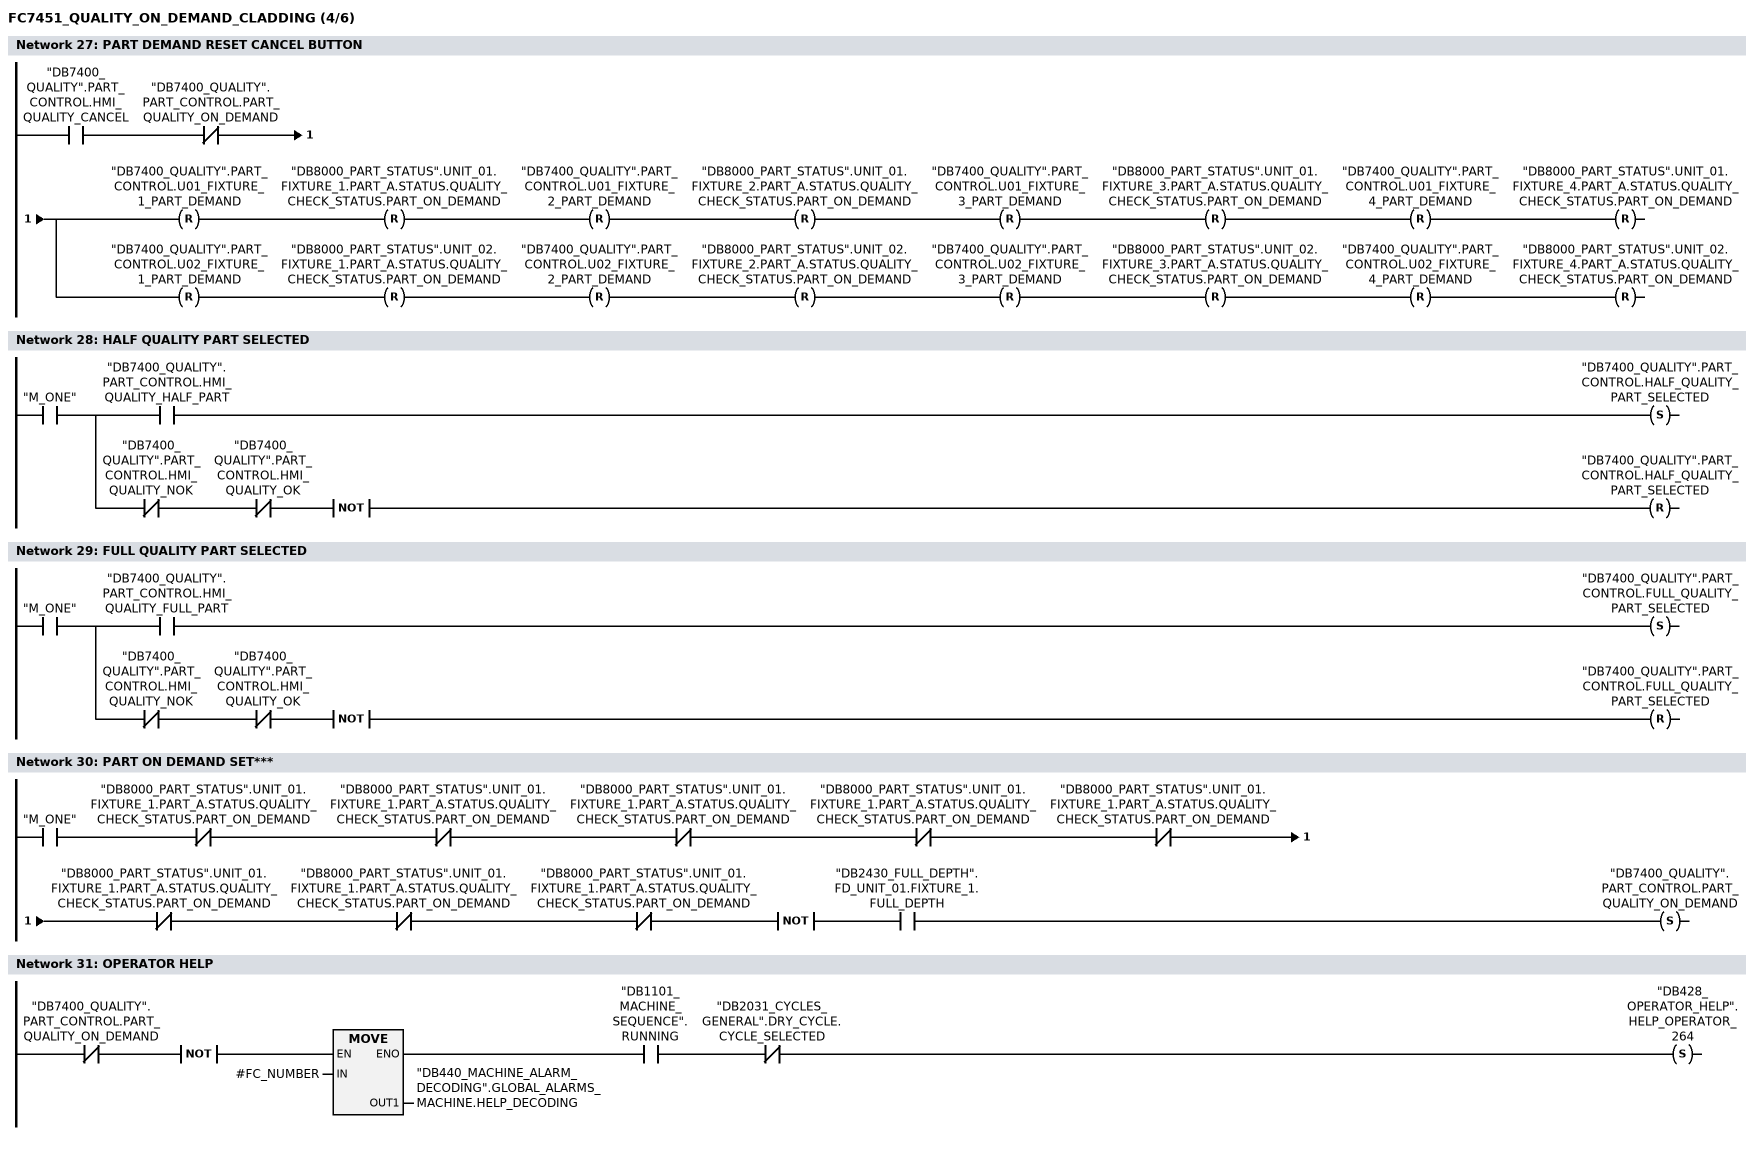
   RUNG wire#powerrail
      Contact( "DB7400_QUALITY".PART_CONTROL.HMI_QUALITY_CANCEL )
      I_Contact( "DB7400_QUALITY".PART_CONTROL.PART_QUALITY_ON_DEMAND )
      wire#w1
      R_Coil( "DB7400_QUALITY".PART_CONTROL.U01_FIXTURE_1_PART_DEMAND )
      R_Coil( "DB8000_PART_STATUS".UNIT_01.FIXTURE_1.PART_A.STATUS.QUALITY_CHECK_STATUS.PART_ON_DEMAND )
      R_Coil( "DB7400_QUALITY".PART_CONTROL.U01_FIXTURE_2_PART_DEMAND )
      R_Coil( "DB8000_PART_STATUS".UNIT_01.FIXTURE_2.PART_A.STATUS.QUALITY_CHECK_STATUS.PART_ON_DEMAND )
      R_Coil( "DB7400_QUALITY".PART_CONTROL.U01_FIXTURE_3_PART_DEMAND )
      R_Coil( "DB8000_PART_STATUS".UNIT_01.FIXTURE_3.PART_A.STATUS.QUALITY_CHECK_STATUS.PART_ON_DEMAND )
      R_Coil( "DB7400_QUALITY".PART_CONTROL.U01_FIXTURE_4_PART_DEMAND )
      R_Coil( "DB8000_PART_STATUS".UNIT_01.FIXTURE_4.PART_A.STATUS.QUALITY_CHECK_STATUS.PART_ON_DEMAND )
   END_RUNG
   RUNG wire#w1
      R_Coil( "DB7400_QUALITY".PART_CONTROL.U02_FIXTURE_1_PART_DEMAND )
      R_Coil( "DB8000_PART_STATUS".UNIT_02.FIXTURE_1.PART_A.STATUS.QUALITY_CHECK_STATUS.PART_ON_DEMAND )
      R_Coil( "DB7400_QUALITY".PART_CONTROL.U02_FIXTURE_2_PART_DEMAND )
      R_Coil( "DB8000_PART_STATUS".UNIT_02.FIXTURE_2.PART_A.STATUS.QUALITY_CHECK_STATUS.PART_ON_DEMAND )
      R_Coil( "DB7400_QUALITY".PART_CONTROL.U02_FIXTURE_3_PART_DEMAND )
      R_Coil( "DB8000_PART_STATUS".UNIT_02.FIXTURE_3.PART_A.STATUS.QUALITY_CHECK_STATUS.PART_ON_DEMAND )
      R_Coil( "DB7400_QUALITY".PART_CONTROL.U02_FIXTURE_4_PART_DEMAND )
      R_Coil( "DB8000_PART_STATUS".UNIT_02.FIXTURE_4.PART_A.STATUS.QUALITY_CHECK_STATUS.PART_ON_DEMAND )
   END_RUNG
   // the same network as SCL:
   IF "DB7400_QUALITY".PART_CONTROL.HMI_QUALITY_CANCEL AND NOT "DB7400_QUALITY".PART_CONTROL.PART_QUALITY_ON_DEMAND THEN
       "DB7400_QUALITY".PART_CONTROL.U01_FIXTURE_1_PART_DEMAND := FALSE;
       "DB8000_PART_STATUS".UNIT_01.FIXTURE_1.PART_A.STATUS.QUALITY_CHECK_STATUS.PART_ON_DEMAND := FALSE;
       "DB7400_QUALITY".PART_CONTROL.U01_FIXTURE_2_PART_DEMAND := FALSE;
       "DB8000_PART_STATUS".UNIT_01.FIXTURE_2.PART_A.STATUS.QUALITY_CHECK_STATUS.PART_ON_DEMAND := FALSE;
       "DB7400_QUALITY".PART_CONTROL.U01_FIXTURE_3_PART_DEMAND := FALSE;
       "DB8000_PART_STATUS".UNIT_01.FIXTURE_3.PART_A.STATUS.QUALITY_CHECK_STATUS.PART_ON_DEMAND := FALSE;
       "DB7400_QUALITY".PART_CONTROL.U01_FIXTURE_4_PART_DEMAND := FALSE;
       "DB8000_PART_STATUS".UNIT_01.FIXTURE_4.PART_A.STATUS.QUALITY_CHECK_STATUS.PART_ON_DEMAND := FALSE;
       "DB7400_QUALITY".PART_CONTROL.U02_FIXTURE_1_PART_DEMAND := FALSE;
       "DB8000_PART_STATUS".UNIT_02.FIXTURE_1.PART_A.STATUS.QUALITY_CHECK_STATUS.PART_ON_DEMAND := FALSE;
       "DB7400_QUALITY".PART_CONTROL.U02_FIXTURE_2_PART_DEMAND := FALSE;
       "DB8000_PART_STATUS".UNIT_02.FIXTURE_2.PART_A.STATUS.QUALITY_CHECK_STATUS.PART_ON_DEMAND := FALSE;
       "DB7400_QUALITY".PART_CONTROL.U02_FIXTURE_3_PART_DEMAND := FALSE;
       "DB8000_PART_STATUS".UNIT_02.FIXTURE_3.PART_A.STATUS.QUALITY_CHECK_STATUS.PART_ON_DEMAND := FALSE;
       "DB7400_QUALITY".PART_CONTROL.U02_FIXTURE_4_PART_DEMAND := FALSE;
       "DB8000_PART_STATUS".UNIT_02.FIXTURE_4.PART_A.STATUS.QUALITY_CHECK_STATUS.PART_ON_DEMAND := FALSE;
   END_IF;
END_REGION

REGION Network 28: HALF QUALITY PART SELECTED
   RUNG wire#powerrail
      Contact( "M_ONE" )
      wire#w1
      Contact( "DB7400_QUALITY".PART_CONTROL.HMI_QUALITY_HALF_PART )
      S_Coil( "DB7400_QUALITY".PART_CONTROL.HALF_QUALITY_PART_SELECTED )
   END_RUNG
   RUNG wire#w1
      I_Contact( "DB7400_QUALITY".PART_CONTROL.HMI_QUALITY_NOK )
      I_Contact( "DB7400_QUALITY".PART_CONTROL.HMI_QUALITY_OK )
      Not()
      R_Coil( "DB7400_QUALITY".PART_CONTROL.HALF_QUALITY_PART_SELECTED )
   END_RUNG
   // the same network as SCL:
   IF "M_ONE" AND "DB7400_QUALITY".PART_CONTROL.HMI_QUALITY_HALF_PART THEN
       "DB7400_QUALITY".PART_CONTROL.HALF_QUALITY_PART_SELECTED := TRUE;
   END_IF;
   IF NOT ("M_ONE" AND NOT "DB7400_QUALITY".PART_CONTROL.HMI_QUALITY_NOK AND NOT "DB7400_QUALITY".PART_CONTROL.HMI_QUALITY_OK) THEN
       "DB7400_QUALITY".PART_CONTROL.HALF_QUALITY_PART_SELECTED := FALSE;
   END_IF;
END_REGION

REGION Network 29: FULL QUALITY PART SELECTED
   RUNG wire#powerrail
      Contact( "M_ONE" )
      wire#w1
      Contact( "DB7400_QUALITY".PART_CONTROL.HMI_QUALITY_FULL_PART )
      S_Coil( "DB7400_QUALITY".PART_CONTROL.FULL_QUALITY_PART_SELECTED )
   END_RUNG
   RUNG wire#w1
      I_Contact( "DB7400_QUALITY".PART_CONTROL.HMI_QUALITY_NOK )
      I_Contact( "DB7400_QUALITY".PART_CONTROL.HMI_QUALITY_OK )
      Not()
      R_Coil( "DB7400_QUALITY".PART_CONTROL.FULL_QUALITY_PART_SELECTED )
   END_RUNG
   // the same network as SCL:
   IF "M_ONE" AND "DB7400_QUALITY".PART_CONTROL.HMI_QUALITY_FULL_PART THEN
       "DB7400_QUALITY".PART_CONTROL.FULL_QUALITY_PART_SELECTED := TRUE;
   END_IF;
   IF NOT ("M_ONE" AND NOT "DB7400_QUALITY".PART_CONTROL.HMI_QUALITY_NOK AND NOT "DB7400_QUALITY".PART_CONTROL.HMI_QUALITY_OK) THEN
       "DB7400_QUALITY".PART_CONTROL.FULL_QUALITY_PART_SELECTED := FALSE;
   END_IF;
END_REGION

REGION Network 30: PART ON DEMAND SET***
   RUNG wire#powerrail
      Contact( "M_ONE" )
      I_Contact( "DB8000_PART_STATUS".UNIT_01.FIXTURE_1.PART_A.STATUS.QUALITY_CHECK_STATUS.PART_ON_DEMAND )
      I_Contact( "DB8000_PART_STATUS".UNIT_01.FIXTURE_1.PART_A.STATUS.QUALITY_CHECK_STATUS.PART_ON_DEMAND )
      I_Contact( "DB8000_PART_STATUS".UNIT_01.FIXTURE_1.PART_A.STATUS.QUALITY_CHECK_STATUS.PART_ON_DEMAND )
      I_Contact( "DB8000_PART_STATUS".UNIT_01.FIXTURE_1.PART_A.STATUS.QUALITY_CHECK_STATUS.PART_ON_DEMAND )
      I_Contact( "DB8000_PART_STATUS".UNIT_01.FIXTURE_1.PART_A.STATUS.QUALITY_CHECK_STATUS.PART_ON_DEMAND )
      I_Contact( "DB8000_PART_STATUS".UNIT_01.FIXTURE_1.PART_A.STATUS.QUALITY_CHECK_STATUS.PART_ON_DEMAND )
      I_Contact( "DB8000_PART_STATUS".UNIT_01.FIXTURE_1.PART_A.STATUS.QUALITY_CHECK_STATUS.PART_ON_DEMAND )
      I_Contact( "DB8000_PART_STATUS".UNIT_01.FIXTURE_1.PART_A.STATUS.QUALITY_CHECK_STATUS.PART_ON_DEMAND )
      Not()
      Contact( "DB2430_FULL_DEPTH".FD_UNIT_01.FIXTURE_1.FULL_DEPTH )
      S_Coil( "DB7400_QUALITY".PART_CONTROL.PART_QUALITY_ON_DEMAND )
   END_RUNG
   // the same network as SCL:
   IF NOT ("M_ONE" AND NOT "DB8000_PART_STATUS".UNIT_01.FIXTURE_1.PART_A.STATUS.QUALITY_CHECK_STATUS.PART_ON_DEMAND AND NOT "DB8000_PART_STATUS".UNIT_01.FIXTURE_1.PART_A.STATUS.QUALITY_CHECK_STATUS.PART_ON_DEMAND AND NOT "DB8000_PART_STATUS".UNIT_01.FIXTURE_1.PART_A.STATUS.QUALITY_CHECK_STATUS.PART_ON_DEMAND AND NOT "DB8000_PART_STATUS".UNIT_01.FIXTURE_1.PART_A.STATUS.QUALITY_CHECK_STATUS.PART_ON_DEMAND AND NOT "DB8000_PART_STATUS".UNIT_01.FIXTURE_1.PART_A.STATUS.QUALITY_CHECK_STATUS.PART_ON_DEMAND AND NOT "DB8000_PART_STATUS".UNIT_01.FIXTURE_1.PART_A.STATUS.QUALITY_CHECK_STATUS.PART_ON_DEMAND AND NOT "DB8000_PART_STATUS".UNIT_01.FIXTURE_1.PART_A.STATUS.QUALITY_CHECK_STATUS.PART_ON_DEMAND AND NOT "DB8000_PART_STATUS".UNIT_01.FIXTURE_1.PART_A.STATUS.QUALITY_CHECK_STATUS.PART_ON_DEMAND) AND "DB2430_FULL_DEPTH".FD_UNIT_01.FIXTURE_1.FULL_DEPTH THEN
       "DB7400_QUALITY".PART_CONTROL.PART_QUALITY_ON_DEMAND := TRUE;
   END_IF;
END_REGION

REGION Network 31: OPERATOR HELP
   RUNG wire#powerrail
      I_Contact( "DB7400_QUALITY".PART_CONTROL.PART_QUALITY_ON_DEMAND )
      Not()
      { S7_GenerateENO := "TRUE" } Move(in := #FC_NUMBER, out1 => "DB440_MACHINE_ALARM_DECODING".GLOBAL_ALARMS_MACHINE.HELP_DECODING)
      Contact( "DB1101_MACHINE_SEQUENCE".RUNNING )
      I_Contact( "DB2031_CYCLES_GENERAL".DRY_CYCLE.CYCLE_SELECTED )
      S_Coil( "DB428_OPERATOR_HELP".HELP_OPERATOR_264 )
   END_RUNG
   // the same network as SCL:
   // ENO of a box is taken as its EN; it also drops when the box reports an error
   #_w1 := NOT (NOT "DB7400_QUALITY".PART_CONTROL.PART_QUALITY_ON_DEMAND);
   IF #_w1 THEN "DB440_MACHINE_ALARM_DECODING".GLOBAL_ALARMS_MACHINE.HELP_DECODING := #FC_NUMBER; END_IF;
   IF #_w1 AND "DB1101_MACHINE_SEQUENCE".RUNNING AND NOT "DB2031_CYCLES_GENERAL".DRY_CYCLE.CYCLE_SELECTED THEN
       "DB428_OPERATOR_HELP".HELP_OPERATOR_264 := TRUE;
   END_IF;
END_REGION

REGION Network 32: PART ON DEMAND RESET
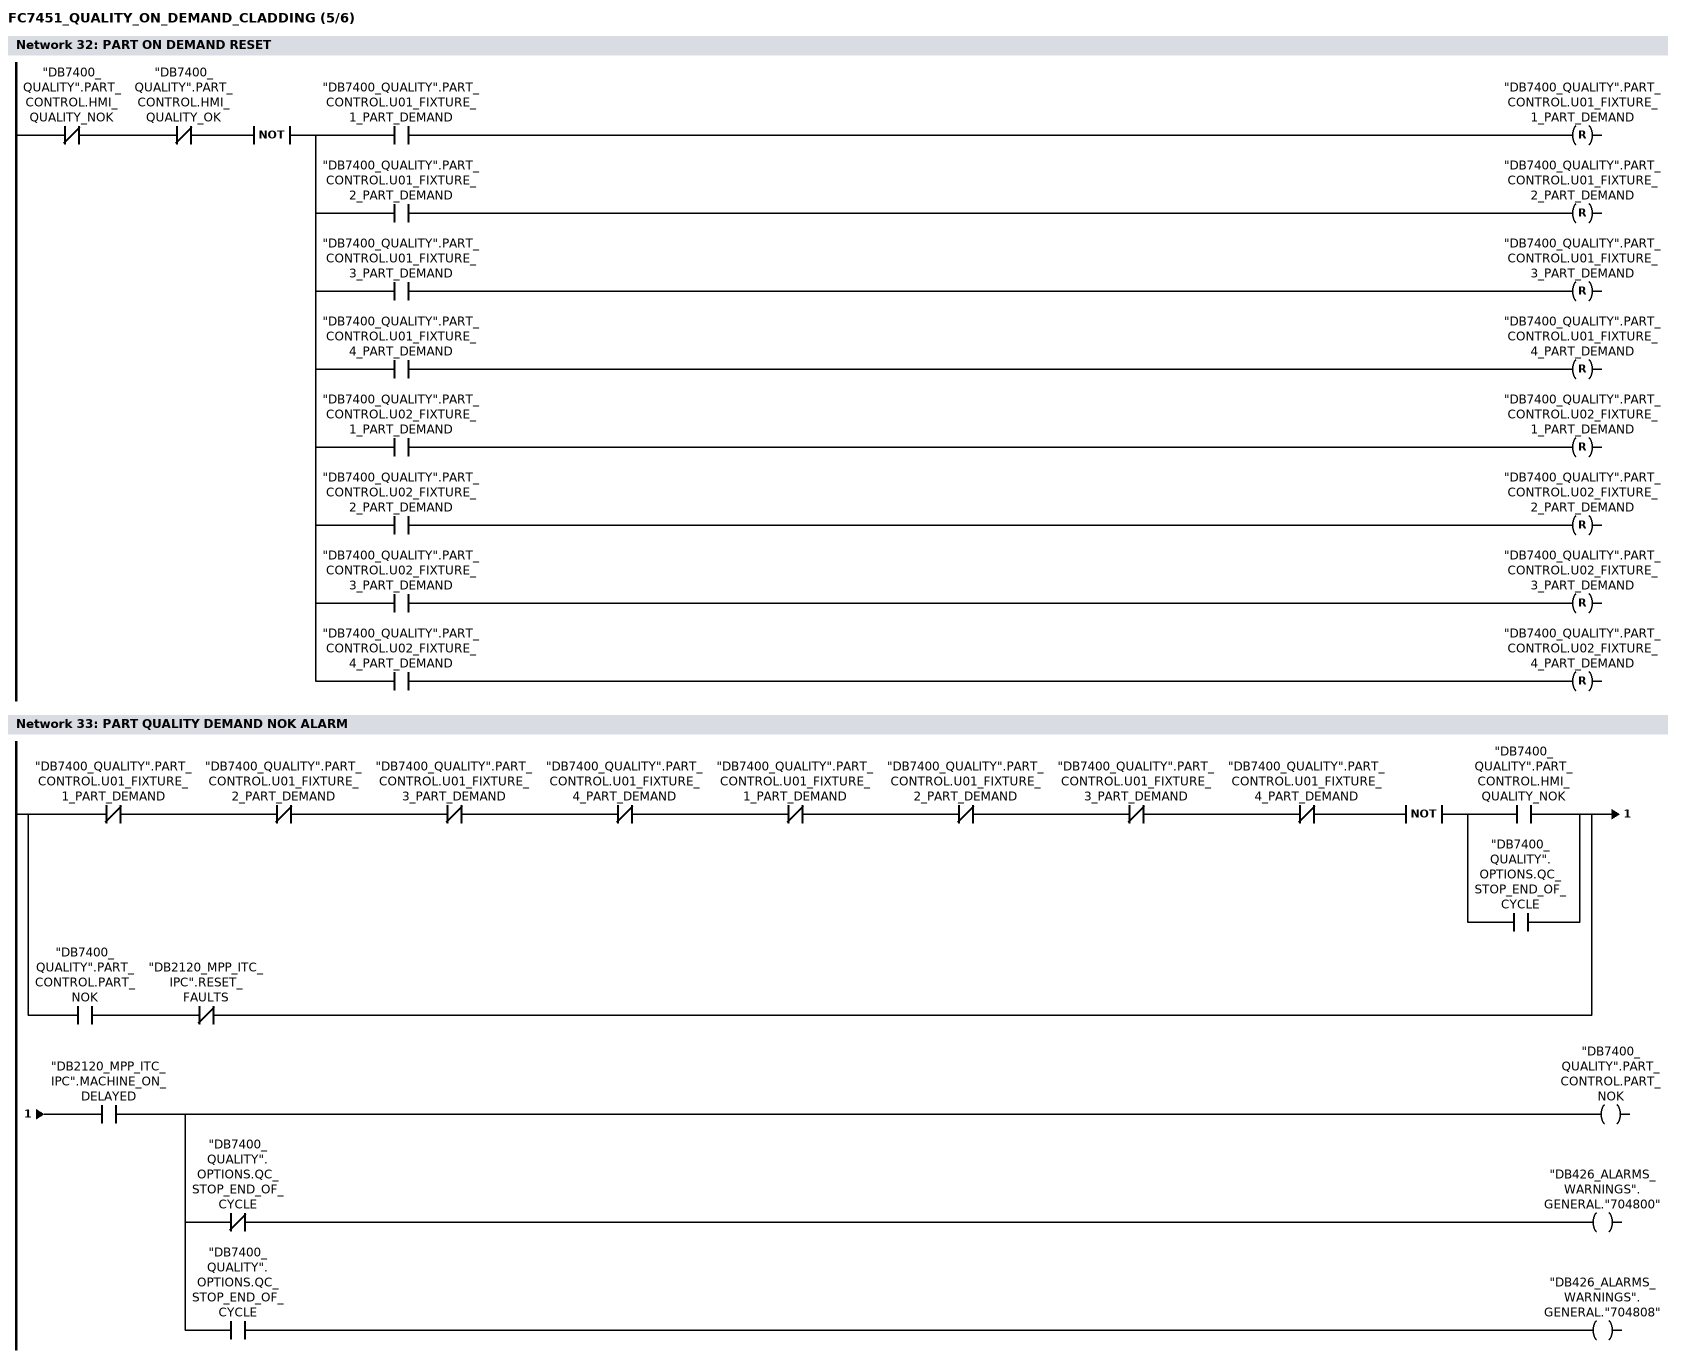
   RUNG wire#powerrail
      I_Contact( "DB7400_QUALITY".PART_CONTROL.HMI_QUALITY_NOK )
      I_Contact( "DB7400_QUALITY".PART_CONTROL.HMI_QUALITY_OK )
      Not()
      wire#w1
      Contact( "DB7400_QUALITY".PART_CONTROL.U01_FIXTURE_1_PART_DEMAND )
      R_Coil( "DB7400_QUALITY".PART_CONTROL.U01_FIXTURE_1_PART_DEMAND )
   END_RUNG
   RUNG wire#w1
      Contact( "DB7400_QUALITY".PART_CONTROL.U01_FIXTURE_2_PART_DEMAND )
      R_Coil( "DB7400_QUALITY".PART_CONTROL.U01_FIXTURE_2_PART_DEMAND )
   END_RUNG
   RUNG wire#w1
      Contact( "DB7400_QUALITY".PART_CONTROL.U01_FIXTURE_3_PART_DEMAND )
      R_Coil( "DB7400_QUALITY".PART_CONTROL.U01_FIXTURE_3_PART_DEMAND )
   END_RUNG
   RUNG wire#w1
      Contact( "DB7400_QUALITY".PART_CONTROL.U01_FIXTURE_4_PART_DEMAND )
      R_Coil( "DB7400_QUALITY".PART_CONTROL.U01_FIXTURE_4_PART_DEMAND )
   END_RUNG
   RUNG wire#w1
      Contact( "DB7400_QUALITY".PART_CONTROL.U02_FIXTURE_1_PART_DEMAND )
      R_Coil( "DB7400_QUALITY".PART_CONTROL.U02_FIXTURE_1_PART_DEMAND )
   END_RUNG
   RUNG wire#w1
      Contact( "DB7400_QUALITY".PART_CONTROL.U02_FIXTURE_2_PART_DEMAND )
      R_Coil( "DB7400_QUALITY".PART_CONTROL.U02_FIXTURE_2_PART_DEMAND )
   END_RUNG
   RUNG wire#w1
      Contact( "DB7400_QUALITY".PART_CONTROL.U02_FIXTURE_3_PART_DEMAND )
      R_Coil( "DB7400_QUALITY".PART_CONTROL.U02_FIXTURE_3_PART_DEMAND )
   END_RUNG
   RUNG wire#w1
      Contact( "DB7400_QUALITY".PART_CONTROL.U02_FIXTURE_4_PART_DEMAND )
      R_Coil( "DB7400_QUALITY".PART_CONTROL.U02_FIXTURE_4_PART_DEMAND )
   END_RUNG
   // the same network as SCL:
   #_w1 := NOT (NOT "DB7400_QUALITY".PART_CONTROL.HMI_QUALITY_NOK AND NOT "DB7400_QUALITY".PART_CONTROL.HMI_QUALITY_OK);
   IF #_w1 AND "DB7400_QUALITY".PART_CONTROL.U01_FIXTURE_1_PART_DEMAND THEN
       "DB7400_QUALITY".PART_CONTROL.U01_FIXTURE_1_PART_DEMAND := FALSE;
   END_IF;
   IF #_w1 AND "DB7400_QUALITY".PART_CONTROL.U01_FIXTURE_2_PART_DEMAND THEN
       "DB7400_QUALITY".PART_CONTROL.U01_FIXTURE_2_PART_DEMAND := FALSE;
   END_IF;
   IF #_w1 AND "DB7400_QUALITY".PART_CONTROL.U01_FIXTURE_3_PART_DEMAND THEN
       "DB7400_QUALITY".PART_CONTROL.U01_FIXTURE_3_PART_DEMAND := FALSE;
   END_IF;
   IF #_w1 AND "DB7400_QUALITY".PART_CONTROL.U01_FIXTURE_4_PART_DEMAND THEN
       "DB7400_QUALITY".PART_CONTROL.U01_FIXTURE_4_PART_DEMAND := FALSE;
   END_IF;
   IF #_w1 AND "DB7400_QUALITY".PART_CONTROL.U02_FIXTURE_1_PART_DEMAND THEN
       "DB7400_QUALITY".PART_CONTROL.U02_FIXTURE_1_PART_DEMAND := FALSE;
   END_IF;
   IF #_w1 AND "DB7400_QUALITY".PART_CONTROL.U02_FIXTURE_2_PART_DEMAND THEN
       "DB7400_QUALITY".PART_CONTROL.U02_FIXTURE_2_PART_DEMAND := FALSE;
   END_IF;
   IF #_w1 AND "DB7400_QUALITY".PART_CONTROL.U02_FIXTURE_3_PART_DEMAND THEN
       "DB7400_QUALITY".PART_CONTROL.U02_FIXTURE_3_PART_DEMAND := FALSE;
   END_IF;
   IF #_w1 AND "DB7400_QUALITY".PART_CONTROL.U02_FIXTURE_4_PART_DEMAND THEN
       "DB7400_QUALITY".PART_CONTROL.U02_FIXTURE_4_PART_DEMAND := FALSE;
   END_IF;
END_REGION

REGION Network 33: PART QUALITY DEMAND NOK ALARM
   RUNG wire#powerrail
      I_Contact( "DB7400_QUALITY".PART_CONTROL.U01_FIXTURE_1_PART_DEMAND )
      I_Contact( "DB7400_QUALITY".PART_CONTROL.U01_FIXTURE_2_PART_DEMAND )
      I_Contact( "DB7400_QUALITY".PART_CONTROL.U01_FIXTURE_3_PART_DEMAND )
      I_Contact( "DB7400_QUALITY".PART_CONTROL.U01_FIXTURE_4_PART_DEMAND )
      I_Contact( "DB7400_QUALITY".PART_CONTROL.U01_FIXTURE_1_PART_DEMAND )
      I_Contact( "DB7400_QUALITY".PART_CONTROL.U01_FIXTURE_2_PART_DEMAND )
      I_Contact( "DB7400_QUALITY".PART_CONTROL.U01_FIXTURE_3_PART_DEMAND )
      I_Contact( "DB7400_QUALITY".PART_CONTROL.U01_FIXTURE_4_PART_DEMAND )
      Not()
      wire#w1
      Contact( "DB7400_QUALITY".PART_CONTROL.HMI_QUALITY_NOK )
      wire#w2
      Contact( "DB2120_MPP_ITC_IPC".MACHINE_ON_DELAYED )
      wire#w3
      Coil( "DB7400_QUALITY".PART_CONTROL.PART_NOK )
   END_RUNG
   RUNG wire#w1
      Contact( "DB7400_QUALITY".OPTIONS.QC_STOP_END_OF_CYCLE )
   END_RUNG wire#w2
   RUNG wire#powerrail
      Contact( "DB7400_QUALITY".PART_CONTROL.PART_NOK )
      I_Contact( "DB2120_MPP_ITC_IPC".RESET_FAULTS )
   END_RUNG wire#w2
   RUNG wire#w3
      I_Contact( "DB7400_QUALITY".OPTIONS.QC_STOP_END_OF_CYCLE )
      Coil( "DB426_ALARMS_WARNINGS".GENERAL."704800" )
   END_RUNG
   RUNG wire#w3
      Contact( "DB7400_QUALITY".OPTIONS.QC_STOP_END_OF_CYCLE )
      Coil( "DB426_ALARMS_WARNINGS".GENERAL."704808" )
   END_RUNG
   // the same network as SCL:
   "DB7400_QUALITY".PART_CONTROL.PART_NOK := ((NOT (NOT "DB7400_QUALITY".PART_CONTROL.U01_FIXTURE_1_PART_DEMAND AND NOT "DB7400_QUALITY".PART_CONTROL.U01_FIXTURE_2_PART_DEMAND AND NOT "DB7400_QUALITY".PART_CONTROL.U01_FIXTURE_3_PART_DEMAND AND NOT "DB7400_QUALITY".PART_CONTROL.U01_FIXTURE_4_PART_DEMAND AND NOT "DB7400_QUALITY".PART_CONTROL.U01_FIXTURE_1_PART_DEMAND AND NOT "DB7400_QUALITY".PART_CONTROL.U01_FIXTURE_2_PART_DEMAND AND NOT "DB7400_QUALITY".PART_CONTROL.U01_FIXTURE_3_PART_DEMAND AND NOT "DB7400_QUALITY".PART_CONTROL.U01_FIXTURE_4_PART_DEMAND) AND ("DB7400_QUALITY".PART_CONTROL.HMI_QUALITY_NOK OR "DB7400_QUALITY".OPTIONS.QC_STOP_END_OF_CYCLE)) OR ("DB7400_QUALITY".PART_CONTROL.PART_NOK AND NOT "DB2120_MPP_ITC_IPC".RESET_FAULTS)) AND "DB2120_MPP_ITC_IPC".MACHINE_ON_DELAYED;
   "DB426_ALARMS_WARNINGS".GENERAL."704800" := "DB7400_QUALITY".PART_CONTROL.PART_NOK AND NOT "DB7400_QUALITY".OPTIONS.QC_STOP_END_OF_CYCLE;
   "DB426_ALARMS_WARNINGS".GENERAL."704808" := "DB7400_QUALITY".PART_CONTROL.PART_NOK AND "DB7400_QUALITY".OPTIONS.QC_STOP_END_OF_CYCLE;
END_REGION

REGION Network 34: RETURN HOME POSITION AND STOP END OF CYCLE ALARMS
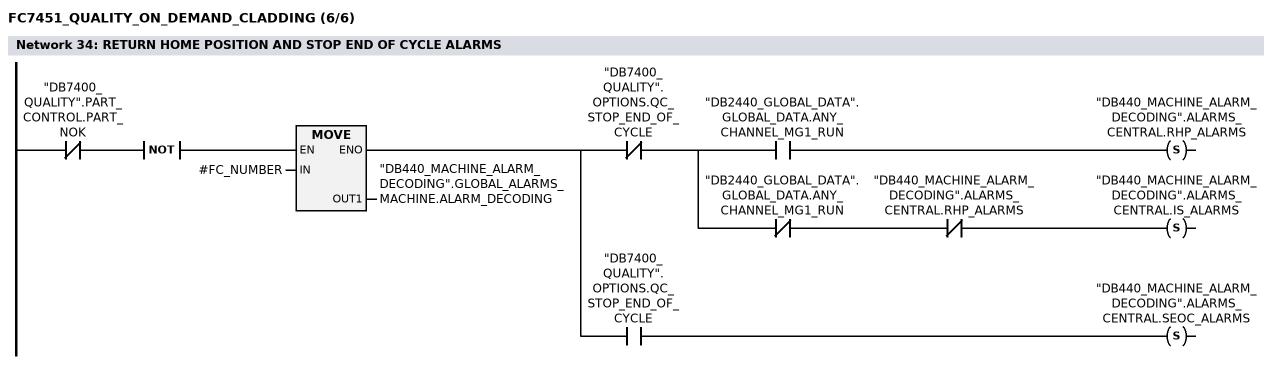
   RUNG wire#powerrail
      I_Contact( "DB7400_QUALITY".PART_CONTROL.PART_NOK )
      Not()
      { S7_GenerateENO := "TRUE" } Move(in := #FC_NUMBER, out1 => "DB440_MACHINE_ALARM_DECODING".GLOBAL_ALARMS_MACHINE.ALARM_DECODING)
      wire#w1
      I_Contact( "DB7400_QUALITY".OPTIONS.QC_STOP_END_OF_CYCLE )
      wire#w2
      Contact( "DB2440_GLOBAL_DATA".GLOBAL_DATA.ANY_CHANNEL_MG1_RUN )
      S_Coil( "DB440_MACHINE_ALARM_DECODING".ALARMS_CENTRAL.RHP_ALARMS )
   END_RUNG
   RUNG wire#w2
      I_Contact( "DB2440_GLOBAL_DATA".GLOBAL_DATA.ANY_CHANNEL_MG1_RUN )
      I_Contact( "DB440_MACHINE_ALARM_DECODING".ALARMS_CENTRAL.RHP_ALARMS )
      S_Coil( "DB440_MACHINE_ALARM_DECODING".ALARMS_CENTRAL.IS_ALARMS )
   END_RUNG
   RUNG wire#w1
      Contact( "DB7400_QUALITY".OPTIONS.QC_STOP_END_OF_CYCLE )
      S_Coil( "DB440_MACHINE_ALARM_DECODING".ALARMS_CENTRAL.SEOC_ALARMS )
   END_RUNG
   // the same network as SCL:
   // ENO of a box is taken as its EN; it also drops when the box reports an error
   #_w1 := NOT (NOT "DB7400_QUALITY".PART_CONTROL.PART_NOK);
   IF #_w1 THEN "DB440_MACHINE_ALARM_DECODING".GLOBAL_ALARMS_MACHINE.ALARM_DECODING := #FC_NUMBER; END_IF;
   #_w2 := #_w1 AND NOT "DB7400_QUALITY".OPTIONS.QC_STOP_END_OF_CYCLE;
   IF #_w2 AND "DB2440_GLOBAL_DATA".GLOBAL_DATA.ANY_CHANNEL_MG1_RUN THEN
       "DB440_MACHINE_ALARM_DECODING".ALARMS_CENTRAL.RHP_ALARMS := TRUE;
   END_IF;
   IF #_w2 AND NOT "DB2440_GLOBAL_DATA".GLOBAL_DATA.ANY_CHANNEL_MG1_RUN AND NOT "DB440_MACHINE_ALARM_DECODING".ALARMS_CENTRAL.RHP_ALARMS THEN
       "DB440_MACHINE_ALARM_DECODING".ALARMS_CENTRAL.IS_ALARMS := TRUE;
   END_IF;
   IF #_w1 AND "DB7400_QUALITY".OPTIONS.QC_STOP_END_OF_CYCLE THEN
       "DB440_MACHINE_ALARM_DECODING".ALARMS_CENTRAL.SEOC_ALARMS := TRUE;
   END_IF;
END_REGION
END_FUNCTION
